// TIA Portal V18 export
TYPE "ST_KeyenceCheckerIV3"
// stored: IsFailsafeCompliant false
   STRUCT
      Common : Struct   // 通用变量
         nID : Int;   // 设备编号
         nMode : Int;   // 控制模式
         bEnable : Bool;   // 启动条件
         bError : Bool;   // 错误
         bWarning : Bool;   // 警告
         bReset : Bool;   // 复位
         bDone : Bool;   // 执行动作完成
         bScreenActive : Bool;   // 激活屏幕
         nModeSwitch : Int;   // 设备操作模式
         nErrorNo : Int;   // 错误代码
         nWarningNo : Int;   // 警告代码
         nLastStep : Int;   // 上一步号
         nCurrentStep : Int;   // 当前步号
         nNextStep : Int;   // 下一步号
         tMaxProcessTime : Time;   // 最大执行时间
         tActProcessTime : Time;   // 实际流程时间
      END_STRUCT;
      In : Struct   // PLC输入变量
         CommandStatus : Struct   // 命令状态
            bTriggerResponse : Bool;   // 触发响应
            bMasterImageRegistration : Bool;   // 主控注册响应
            bProgramSwitchingResponse : Bool;   // 程序切换响应
            bWarningClearResponse : Bool;   // 警报清除响应
            bStatisticsResetResponse : Bool;   // 统计复位响应
            bBufferClearResponse : Bool;   // 缓存清除响应
            bSDCardStopSaveResponse : Bool;   // SD卡保存停止响应
            bChangeParameterResponse : Bool;   // 设定值更改响应
            bTriggerFailed : Bool;   // 触发失败
            bMasterImageRegistrationFailed : Bool;   // 主控注册失败
            bProgramSwitchingFailed : Bool;   // 程序切换失败
            bReserved1 : Bool;   // 系统预约
            bReserved2 : Bool;   // 系统预约
            bReserved3 : Bool;   // 系统预约
            bSDCardStopSaveFailed : Bool;   // SD 卡保存停止失败
            bChangeParameterFailed : Bool;   // 设定值更改失败
            bResultAvailable : Bool;   // 可获取结果
            bResultUpdateComplete : Bool;   // 结果更新完成
            bBusy : Bool;   // BUSY
            bImaging : Bool;   // 拍摄状态
            bRun : Bool;   // 运行
            bReady : Bool;   // 就绪
            bReserved4 : Bool;   // 系统预约
            bSDCardStatus : Bool;   // SD 卡识别状态
            bClassificationModeInformation : Bool;   // 分类模式信息
            bReserved5 : Bool;   // 系统预约
            bReserved6 : Bool;   // 系统预约
            bReserved7 : Bool;   // 系统预约
            bSDCardStorageShortage : Bool;   // SD 卡容量不足
            bBufferOverrun : Bool;   // 缓存溢出
            bWarning : Bool;   // 警报
            bError : Bool;   // 错误
         END_STRUCT;
         DeviceResults : Struct   // 设备结果
            bOverallJudgmentOK : Bool;   // 综合判断OK
            bPositionCorrection : Bool;   // 位置修正
            bLogic1 : Bool;   // LOGIC1
            bLogic2 : Bool;   // LOGIC2
            bLogic3 : Bool;   // LOGIC3
            bLogic4 : Bool;   // LOGIC4
            bOverallJudgmentNG : Bool;   // 综合判断NG
            bReserved1 : Bool;   // 系统预约
            nReserved2 : Byte;   // 系统预约
            aToolResult : Array[1..16] of Bool;   // 单个工具的好坏
         END_STRUCT;
         "DeviceStatus" : Struct   // 设备状态
            nErrorNo : Word;   // 错误编号（无符号 16bit 数据）
            nWarningNo : Word;   // 警报编号（无符号 16bit 数据）
            nNumberOfRemainingBuffers : Word;   // 剩余缓存数（无符号 16bit 数据）
            nChecksum : Word;   // 设定检查和（无符号 16bit 数据）
            nCurrentProgramNo : Word;   // 当前程序编号（无符号 16bit 数据）
            nProgramNoDuringJudgment : Word;   // 判断时程序编号（无符号 16bit 数据）
            nResultNo : Word;   // 结果编号（无符号 16bit 数据）
            nProcessingtime : Word;   // 处理时间（无符号 16bit 数据）
         END_STRUCT;
         "DeviceStatistics" : Struct   // 设备统计
            nProcessingTimeMAX : Word;   // 处理时间 MAX（无符号 16bit 数据）
            nProcessingTimeMIN : Word;   // 处理时间 MIN（无符号 16bit 数据）
            nProcessingTimeAVE : Word;   // 处理时间 AVE（无符号 16bit 数据）
            nReserved1 : Word;   // 系统预约
            nNumberOfTriggers : DWord;   // 触发次数（无符号 32bit 数据）
            nNumberOfOKs : DWord;   // OK 次数/分类次数（无符号 32bit 数据）
            nNumberOfNGs : DWord;   // NG 次数（无符号 32bit 数据）
            nNumberOfTriggerErrors : DWord;   // 触发错误次数（无符号 32bit 数据）
            nReserved2 : DWord;   // 系统预约
         END_STRUCT;
         "PositionAdjustResult" : Struct   // 位置调整结果
            nPositionCorrectionToolMatchingRate : Word;   // 位置修正分数（无符号 16bit 数据）
            nPositionCorrectionToolMatchingRateMAX : Word;   // 位置修正分数 MAX（无符号 16bit 数据）
            nPositionCorrectionToolMatchingRateMIN : Word;   // 位置修正分数 MIN（无符号 16bit 数据）
            nPositionCorrectionToolThreshold : Word;   // 位置修正分数 下限阈值（无符号 16bit 数据 )
            nReserved1 : Word;   // 系统预约
            nReserved2 : Word := 16#0000;   // 系统预约
            nReserved3 : Word := 16#0000;   // 系统预约
            nReserved4 : Word := 16#0000;   // 系统预约
            nReserved5 : Word := 16#0000;   // 系统预约
            nReserved6 : Word := 16#0000;   // 系统预约
         END_STRUCT;
         ToolResult : Array[1..64] of Struct   // 工具结果
            nToolMatchingRate : Word;   // 工具相似度（无符号 16bit 数据）
            nToolMatchingRateMAX : Word;   // 工具相似度 MAX（无符号 16bit 数据）
            nToolMatchingRateMIN : Word;   // 工具相似度 MIN（无符号 16bit 数据）
            nToolLowerLimitValue : Word;   // 工具 下限阈值（无符号 16bit 数据 )
            nToolUpperLimitValue : Word;   // 工具 上限阈值（无符号 16bit 数据 )
            nDecimalPosition : Word;   // 小数点位置（16bit 无符号整数）
            "nPitchPresentValueMAX/ColorAverageH (hue)" : Word;   // 间距当前值 MAX/ 彩色识别 H（色相）（16 bit 无符号整数）
            "nPitchPresentValueMIN/ColorAverageS(saturation)" : Word;   // 间距当前值 MIN/ 彩色识别 S（彩度）（16 bit 无符号整数）
            "nNumberOfPitches/ColorAverageV(brightness)/BrightnessAverage" : Word;   // 间距数量 / 彩色识别 V（彩度） / 亮度平均 亮度（16 bit 无符号整数）
            nReserved1 : Word;   // 系统预约
         END_STRUCT;
         ExtendedDeviceResult : Struct   // 设备结果标准/分类模式
            nMasterNumber : Word;   // 主控编号（无符号16bit数据）
            aToolResult : Array[17..64] of Bool;   // 单个工具好坏
         END_STRUCT;
      END_STRUCT;
      Out : Struct   // PLC输出变量
         CommandControl : Struct   // 控制请求
            bTriggerRequest : Bool;   // 触发请求
            bMasterRegistrationRequest : Bool;   // 主控注册请求
            bProgramSwitchingRequest : Bool;   // 程序切换请求
            bWarningClearRequest : Bool;   // 警报清除请求
            bStatisticsResetRequest : Bool;   // 统计复位请求
            bBufferClearRequest : Bool;   // 缓存清除请求
            bSDCardSaveStopRequest : Bool;   // SD 卡保存停止请求
            bParameterChangeRequest : Bool;   // 设定值更改请求
            nReserved1 : Byte;   // 系统预约
            bResultAcquisitionCompleteNotification : Bool;   // 结果获取完成通知
            bReserved2 : Bool;   // 系统预约
            bReserved3 : Bool;   // 系统预约
            bReserved4 : Bool;   // 系统预约
            bReserved5 : Bool;   // 系统预约
            bReserved6 : Bool;   // 系统预约
            bReserved7 : Bool;   // 系统预约
            bReserved8 : Bool;   // 系统预约
            nReserved9 : Byte;   // 系统预约
            nProgramNo : Word;   // 程序编号
            nSetNumber : Word;   // 设定值设定编号
            nSetParameter : DWord;   // 设定值
         END_STRUCT;
      END_STRUCT;
      Para : Struct   // 参数变量
         nInAdr1 : HW_IO;   // 输入地址1
         nInAdr2 : HW_IO;   // 输入地址2
         nInAdr3 : HW_IO;   // 输入地址3
         nInAdr4 : HW_IO;   // 输入地址4
         nInAdr5 : HW_IO;   // 输入地址5
         nInAdr6 : HW_IO;   // 输入地址6
         nInAdr7 : HW_IO;   // 输入地址7
         nInAdr8 : HW_IO;   // 输入地址8
         nInAdr9 : HW_IO;   // 输入地址9
         nInAdr10 : HW_IO;   // 输入地址10
         nInAdr11 : HW_IO;   // 输入地址11
         nInAdr12 : HW_IO;   // 输入地址12
         nInAdr13 : HW_IO;   // 输入地址13
         nInAdr14 : HW_IO;   // 输入地址14
         nInAdr15 : HW_IO;   // 输入地址15
         nInAdr16 : HW_IO;   // 输入地址16
         nInAdr17 : HW_IO;   // 输入地址17
         nInAdr18 : HW_IO;   // 输入地址18
         nInAdr19 : HW_IO;   // 输入地址19
         nInAdr20 : HW_IO;   // 输入地址20
         nInAdr21 : HW_IO;   // 输入地址21
         nInAdr22 : HW_IO;   // 输入地址22
         nInAdr23 : HW_IO;   // 输入地址23
         nInAdr24 : HW_IO;   // 输入地址24
         nInAdr25 : HW_IO;   // 输入地址25
         nInAdr26 : HW_IO;   // 输入地址26
         nInAdr27 : HW_IO;   // 输入地址27
         nInAdr28 : HW_IO;   // 输入地址28
         nInAdr29 : HW_IO;   // 输入地址29
         nInAdr30 : HW_IO;   // 输入地址30
         nInAdr31 : HW_IO;   // 输入地址31
         nInAdr32 : HW_IO;   // 输入地址32
         nInAdr33 : HW_IO;   // 输入地址33
         nInAdr34 : HW_IO;   // 输入地址34
         nInAdr35 : HW_IO;   // 输入地址35
         nInAdr36 : HW_IO;   // 输入地址36
         nInAdr37 : HW_IO;   // 输入地址37
         nInAdr38 : HW_IO;   // 输入地址38
         nInAdr39 : HW_IO;   // 输入地址39
         nInAdr40 : HW_IO;   // 输入地址68
         nInAdr41 : HW_IO;   // 输入地址67
         nInAdr42 : HW_IO;   // 输入地址66
         nInAdr43 : HW_IO;   // 输入地址65
         nInAdr44 : HW_IO;   // 输入地址64
         nInAdr45 : HW_IO;   // 输入地址63
         nInAdr46 : HW_IO;   // 输入地址62
         nInAdr47 : HW_IO;   // 输入地址61
         nInAdr48 : HW_IO;   // 输入地址60
         nInAdr49 : HW_IO;   // 输入地址59
         nInAdr50 : HW_IO;   // 输入地址58
         nInAdr51 : HW_IO;   // 输入地址57
         nInAdr52 : HW_IO;   // 输入地址56
         nInAdr53 : HW_IO;   // 输入地址55
         nInAdr54 : HW_IO;   // 输入地址54
         nInAdr55 : HW_IO;   // 输入地址53
         nInAdr56 : HW_IO;   // 输入地址52
         nInAdr57 : HW_IO;   // 输入地址51
         nInAdr58 : HW_IO;   // 输入地址50
         nInAdr59 : HW_IO;   // 输入地址49
         nInAdr60 : HW_IO;   // 输入地址48
         nInAdr61 : HW_IO;   // 输入地址47
         nInAdr62 : HW_IO;   // 输入地址46
         nInAdr63 : HW_IO;   // 输入地址45
         nInAdr64 : HW_IO;   // 输入地址44
         nInAdr65 : HW_IO;   // 输入地址43
         nInAdr66 : HW_IO;   // 输入地址42
         nInAdr67 : HW_IO;   // 输入地址41
         nInAdr68 : HW_IO;   // 输入地址40
         nInAdr69 : HW_IO;   // 输入地址69
         nInAdr70 : HW_IO;   // 输入地址70
         nOutAdr1 : HW_IO;   // 输出地址1
         aToolResult : Array[1..64] of Bool;   // 单个工具的好坏
         aToolResultHMI : Array[1..16] of Byte;   // 单个工具的好坏
         ToolResult : Array[1..64] of Struct   // 工具结果
            nToolMatchingRate : Word;   // 工具相似度（无符号 16bit 数据）
            nToolMatchingRateMAX : Word;   // 工具相似度 MAX（无符号 16bit 数据）
            nToolMatchingRateMIN : Word;   // 工具相似度 MIN（无符号 16bit 数据）
            nToolLowerLimitValue : Word;   // 工具 下限阈值（无符号 16bit 数据 )
            nToolUpperLimitValue : Word;   // 工具 上限阈值（无符号 16bit 数据 )
            nDecimalPosition : Word;   // 小数点位置（16bit 无符号整数）
            "nPitchPresentValueMAX/ColorAverageH (hue)" : Word;   // 间距当前值 MAX/ 彩色识别 H（色相）（16 bit 无符号整数）
            "nPitchPresentValueMIN/ColorAverageS(saturation)" : Word;   // 间距当前值 MIN/ 彩色识别 S（彩度）（16 bit 无符号整数）
            "nNumberOfPitches/ColorAverageV(brightness)/BrightnessAverage" : Word;   // 间距数量 / 彩色识别 V（彩度） / 亮度平均 亮度（16 bit 无符号整数）
            nReserved1 : Word;   // 系统预约
         END_STRUCT;
         nProgramNo : Word;   // 设置程序号
         bProductOverallOK : Bool;   // 产品综合OK
         bProductOverallNG : Bool;   // 产品综合NG
      END_STRUCT;
   END_STRUCT;
END_TYPE
